PROGRAM prgGrid
VAR PERSISTENT
	rSizeGridConn				: REAL;									//{#lynus.ag#()}
END_VAR
VAR
	fbGrid						: FB_Grid_Power_Ext_Input;
	lrGridPower					: LREAL;								//{#lynus.ag#()}
	lrGridPower_Consumption		: LREAL;								//{#lynus.ag#()}
	lrGridPower_Production		: LREAL;								//{#lynus.ag#()}
END_VAR







fbGrid(
	bEnable:= TRUE, 
	diNrOfEMS_IN:= prgEMS.fbEMS.diNrOfEMS_OUT, 
	rSizeGridConn:= rSizeGridConn, 
	bExtErrorGrid:= , 
	lrExtGridPower:= prgEM.lrPower_Grid_TotalkW,	
	lrExtTotalCounterEnergy_Consumption:= 0, 
	lrExtTotalCounterEnergy_Production:= 0, 
	lrExtCounterEnergyT1_Consumption:= 0, 
	lrExtCounterEnergyT2_Consumption:= 0, 
	lrExtCounterEnergyT1_Production:= 0, 
	lrExtCounterEnergyT2_Production:= 0, 
	stDataGrid=> , 
	diNrOfGrid_OUT=> );
	
lrGridPower := fbGrid.stDataGrid.lrPower;
IF lrGridPower >=0 THEN 
	lrGridPower_Consumption := lrGridPower;
	lrGridPower_Production := 0;
ELSE
	lrGridPower_Consumption := 0;
	lrGridPower_Production := -lrGridPower;
END_IF

END_PROGRAM

(* stored: Version 1.1.0.1, ProductVersion 3.1.4024.12
   POU prgGrid: Id {7baeccdf-076f-481e-be2b-3e357576b311}, SpecialFunc None *)
